{attribute 'qualified_only'}
{attribute 'strict'}
{attribute 'to_string'}
TYPE ST105_Cylinders_e :
(
    Ausschieber_ab_auf,
    Ausschieber_vor_zuruck,
    _max
);
END_TYPE

(* stored: Version 1.1.0.1, ProductVersion 3.1.4024.6
   EnumerationTextList ST105_Cylinders_e: Id {b8e722ed-eb2d-4459-871a-3d60416093db} *)
